FUNCTION_BLOCK FB_LamparaIntermitente_ST
// La lampara parpadea de forma continua
VAR_INPUT
    TiempoParpadeo: TIME := T#500MS;
END_VAR
VAR
    Temporizador: TON;
    Lampara AT %Q*: BOOL;
END_VAR

// Temporizador auto-pilotado
Temporizador(
    IN := NOT Temporizador.Q,
    PT := TiempoParpadeo
    );

// Salida conmutada
IF Temporizador.Q THEN
    Lampara := NOT Lampara;
END_IF;

END_FUNCTION_BLOCK

(* stored: Version 1.1.0.1, ProductVersion 3.1.4024.15
   POU FB_LamparaIntermitente_ST: Id {558a93e3-8cb7-48c2-9109-65a38d8c0981}, SpecialFunc None *)
